// TIA Portal project "ft" (V16)

(* hardware
DEVICE "S7-1200 station_1"  S7-1200 Station
   slot 0: "Rack_0"  S7-1200 Rack  Rack  V1.0
   slot 1: "PLC_1"  CPU 1214C DC/DC/DC  6ES7 214-1AG40-0XB0  V4.2
   slot 2: "DI 16/DQ 16x24VDC_1"  6ES7 223-1BL32-0XB0  V2.0
   slot 3: "DI 16/DQ 16x24VDC_2"  6ES7 223-1BL32-0XB0  V2.0
   slot 4: "DI 16/DQ 16x24VDC_3"  6ES7 223-1BL32-0XB0  V2.0
   slot 5: "DI 16/DQ 16x24VDC_4"  6ES7 223-1BL32-0XB0  V2.0
   slot 6: "DI 16/DQ 16x24VDC_5"  6ES7 223-1BL32-0XB0  V2.0
   slot 7: "DI 16/DQ 16x24VDC_6"  6ES7 223-1BL32-0XB0  V2.0
*)

// ===== PLC "PLC_1"  CPU 1214C DC/DC/DC =====

VAR_GLOBAL   // PLC tag table "Input tags_1"
   "IN_1-0.0" AT %I0.0 : Bool;
   "IN_1-0.1" AT %I0.1 : Bool;
   "IN_1-0.2" AT %I0.2 : Bool;
   "IN_1-0.3" AT %I0.3 : Bool;
   "IN_1-0.4" AT %I0.4 : Bool;
   "IN_1-0.5" AT %I0.5 : Bool;
   "IN_1-0.6" AT %I0.6 : Bool;
   "IN_1-0.7" AT %I0.7 : Bool;
   "IN_1-1.0" AT %I1.0 : Bool;
   "IN_1-1.1" AT %I1.1 : Bool;
   "IN_1-1.2" AT %I1.5 : Bool;
   "IN_1-1.3" AT %I1.4 : Bool;
   "IN_1-1.4" AT %I1.3 : Bool;
   "IN_1-1.5" AT %I1.2 : Bool;
   "AN_1" AT %IW64 : Int;
   "AN_2" AT %IW66 : Int;
END_VAR

VAR_GLOBAL   // PLC tag table "Output tags_1"
   "OUT_1-0.0" AT %Q0.0 : Bool;
   "OUT_1-0.1" AT %Q0.1 : Bool;
   "OUT_1-0.2" AT %Q0.2 : Bool;
   "OUT_1-0.3" AT %Q0.3 : Bool;
   "OUT_1-0.4" AT %Q0.4 : Bool;
   "OUT_1-0.5" AT %Q0.5 : Bool;
   "OUT_1-0.6" AT %Q0.6 : Bool;
   "OUT_1-0.7" AT %Q0.7 : Bool;
   "OUT_1-1.0" AT %Q1.0 : Bool;
   "OUT_1-1.1" AT %Q1.1 : Bool;
END_VAR

VAR_GLOBAL   // PLC tag table "Input tags_2"
   "IN_2-0.0" AT %I8.0 : Bool;
   "IN_2-0.1" AT %I8.1 : Bool;
   "IN_2-0.2" AT %I8.2 : Bool;
   "IN_2-0.3" AT %I8.3 : Bool;
   "IN_2-0.4" AT %I8.4 : Bool;
   "IN_2-0.5" AT %I8.5 : Bool;
   "IN_2-0.6" AT %I8.6 : Bool;
   "IN_2-0.7" AT %I8.7 : Bool;
   "IN_2-1.0" AT %I9.0 : Bool;
   "IN_2-1.1" AT %I9.1 : Bool;
   "IN_2-1.2" AT %I9.2 : Bool;
   "IN_2-1.3" AT %I9.3 : Bool;
   "IN_2-1.4" AT %I9.4 : Bool;
   "IN_2-1.5" AT %I9.5 : Bool;
   "IN_2-1.6" AT %I9.6 : Bool;
   "IN_2-1.7" AT %I9.7 : Bool;
END_VAR

VAR_GLOBAL   // PLC tag table "Output tags_2"
   "OUT_2-0.0" AT %Q8.0 : Bool;
   "OUT_2-0.1" AT %Q8.1 : Bool;
   "OUT_2-0.2" AT %Q8.2 : Bool;
   "OUT_2-0.3" AT %Q8.3 : Bool;
   "OUT_2-0.4" AT %Q8.4 : Bool;
   "OUT_2-0.5" AT %Q8.5 : Bool;
   "OUT_2-0.6" AT %Q8.6 : Bool;
   "OUT_2-0.7" AT %Q8.7 : Bool;
   "OUT_2-1.0" AT %Q9.0 : Bool;
   "OUT_2-1.1" AT %Q9.1 : Bool;
   "OUT_2-1.2" AT %Q9.2 : Bool;
   "OUT_2-1.3" AT %Q9.3 : Bool;
   "OUT_2-1.4" AT %Q9.4 : Bool;
   "OUT_2-1.5" AT %Q9.5 : Bool;
   "OUT_2-1.6" AT %Q9.6 : Bool;
   "OUT_2-1.7" AT %Q9.7 : Bool;
END_VAR

VAR_GLOBAL   // PLC tag table "Input tags_3"
   "IN_3-0.0" AT %I12.0 : Bool;
   "IN_3-0.1" AT %I12.1 : Bool;
   "IN_3-0.2" AT %I12.2 : Bool;
   "IN_3-0.3" AT %I12.3 : Bool;
   "IN_3-0.4" AT %I12.4 : Bool;
   "IN_3-0.5" AT %I12.5 : Bool;
   "IN_3-0.6" AT %I12.6 : Bool;
   "IN_3-0.7" AT %I12.7 : Bool;
   "IN_3-1.0" AT %I13.0 : Bool;
   "IN_3-1.1" AT %I13.1 : Bool;
   "IN_3-1.2" AT %I13.2 : Bool;
   "IN_3-1.3" AT %I13.3 : Bool;
   "IN_3-1.4" AT %I13.4 : Bool;
   "IN_3-1.5" AT %I13.5 : Bool;
   "IN_3-1.6" AT %I13.6 : Bool;
   "IN_3-1.7" AT %I13.7 : Bool;
END_VAR

VAR_GLOBAL   // PLC tag table "Output tags_3"
   "OUT_3-0.0" AT %Q12.0 : Bool;
   "OUT_3-0.1" AT %Q12.1 : Bool;
   "OUT_3-0.2" AT %Q12.2 : Bool;
   "OUT_3-0.3" AT %Q12.3 : Bool;
   "OUT_3-0.4" AT %Q12.4 : Bool;
   "OUT_3-0.5" AT %Q12.5 : Bool;
   "OUT_3-0.6" AT %Q12.6 : Bool;
   "OUT_3-0.7" AT %Q12.7 : Bool;
   "OUT_3-1.0" AT %Q13.0 : Bool;
   "OUT_3-1.1" AT %Q13.1 : Bool;
   "OUT_3-1.2" AT %Q13.2 : Bool;
   "OUT_3-1.3" AT %Q13.3 : Bool;
   "OUT_3-1.4" AT %Q13.4 : Bool;
   "OUT_3-1.5" AT %Q13.5 : Bool;
   "OUT_3-1.6" AT %Q13.6 : Bool;
   "OUT_3-1.7" AT %Q13.7 : Bool;
END_VAR

VAR_GLOBAL   // PLC tag table "Input tags_4"
   "IN_4-0.0" AT %I16.0 : Bool;
   "IN_4-0.1" AT %I16.1 : Bool;
   "IN_4-0.2" AT %I16.2 : Bool;
   "IN_4-0.3" AT %I16.3 : Bool;
   "IN_4-0.4" AT %I16.4 : Bool;
   "IN_4-0.5" AT %I16.5 : Bool;
   "IN_4-0.6" AT %I16.6 : Bool;
   "IN_4-0.7" AT %I16.7 : Bool;
   "IN_4-1.0" AT %I17.0 : Bool;
   "IN_4-1.1" AT %I17.1 : Bool;
   "IN_4-1.2" AT %I17.2 : Bool;
   "IN_4-1.3" AT %I17.3 : Bool;
   "IN_4-1.4" AT %I17.4 : Bool;
   "IN_4-1.5" AT %I17.5 : Bool;
   "IN_4-1.6" AT %I17.6 : Bool;
   "IN_4-1.7" AT %I17.7 : Bool;
END_VAR

VAR_GLOBAL   // PLC tag table "Output tags_4"
   "OUT_4-0.0" AT %Q16.0 : Bool;
   "OUT_4-0.1" AT %Q16.1 : Bool;
   "OUT_4-0.2" AT %Q16.2 : Bool;
   "OUT_4-0.3" AT %Q16.3 : Bool;
   "OUT_4-0.4" AT %Q16.4 : Bool;
   "OUT_4-0.5" AT %Q16.5 : Bool;
   "OUT_4-0.6" AT %Q16.6 : Bool;
   "OUT_4-0.7" AT %Q16.7 : Bool;
   "OUT_4-1.0" AT %Q17.0 : Bool;
   "OUT_4-1.1" AT %Q17.1 : Bool;
   "OUT_4-1.2" AT %Q17.2 : Bool;
   "OUT_4-1.3" AT %Q17.3 : Bool;
   "OUT_4-1.4" AT %Q17.4 : Bool;
   "OUT_4-1.5" AT %Q17.5 : Bool;
   "OUT_4-1.6" AT %Q17.6 : Bool;
   "OUT_4-1.7" AT %Q17.7 : Bool;
END_VAR

VAR_GLOBAL   // PLC tag table "Input tags_5"
   "IN_5-0.0" AT %I20.0 : Bool;
   "IN_5-0.1" AT %I20.1 : Bool;
   "IN_5-0.2" AT %I20.2 : Bool;
   "IN_5-0.3" AT %I20.3 : Bool;
   "IN_5-0.4" AT %I20.4 : Bool;
   "IN_5-0.5" AT %I20.5 : Bool;
   "IN_5-0.6" AT %I20.6 : Bool;
   "IN_5-0.7" AT %I20.7 : Bool;
   "IN_5-1.0" AT %I21.0 : Bool;
   "IN_5-1.1" AT %I21.1 : Bool;
   "IN_5-1.2" AT %I21.2 : Bool;
   "IN_5-1.3" AT %I21.3 : Bool;
   "IN_5-1.4" AT %I21.4 : Bool;
   "IN_5-1.5" AT %I21.5 : Bool;
   "IN_5-1.6" AT %I21.6 : Bool;
   "IN_5-1.7" AT %I21.7 : Bool;
END_VAR

VAR_GLOBAL   // PLC tag table "Output tags_5"
   "OUT_5-0.0" AT %Q20.0 : Bool;
   "OUT_5-0.1" AT %Q20.1 : Bool;
   "OUT_5-0.2" AT %Q20.2 : Bool;
   "OUT_5-0.3" AT %Q20.3 : Bool;
   "OUT_5-0.4" AT %Q20.4 : Bool;
   "OUT_5-0.5" AT %Q20.5 : Bool;
   "OUT_5-0.6" AT %Q20.6 : Bool;
   "OUT_5-0.7" AT %Q20.7 : Bool;
   "OUT_5-1.0" AT %Q21.0 : Bool;
   "OUT_5-1.1" AT %Q21.1 : Bool;
   "OUT_5-1.2" AT %Q21.2 : Bool;
   "OUT_5-1.3" AT %Q21.3 : Bool;
   "OUT_5-1.4" AT %Q21.4 : Bool;
   "OUT_5-1.5" AT %Q21.5 : Bool;
   "OUT_5-1.6" AT %Q21.6 : Bool;
   "OUT_5-1.7" AT %Q21.7 : Bool;
END_VAR

VAR_GLOBAL   // PLC tag table "Input tags_6"
   "IN_6-0.0" AT %I24.0 : Bool;
   "IN_6-0.1" AT %I24.1 : Bool;
   "IN_6-0.2" AT %I24.2 : Bool;
   "IN_6-0.3" AT %I24.3 : Bool;
   "IN_6-0.4" AT %I24.4 : Bool;
   "IN_6-0.5" AT %I24.5 : Bool;
   "IN_6-0.6" AT %I24.6 : Bool;
   "IN_6-0.7" AT %I24.7 : Bool;
   "IN_6-1.0" AT %I25.0 : Bool;
   "IN_6-1.1" AT %I25.1 : Bool;
   "IN_6-1.2" AT %I25.2 : Bool;
   "IN_6-1.3" AT %I25.3 : Bool;
   "IN_6-1.4" AT %I25.4 : Bool;
   "IN_6-1.5" AT %I25.5 : Bool;
   "IN_6-1.6" AT %I25.6 : Bool;
   "IN_6-1.7" AT %I25.7 : Bool;
END_VAR

VAR_GLOBAL   // PLC tag table "Output tags_6"
   "OUT_6-0.0" AT %Q24.0 : Bool;
   "OUT_6-0.1" AT %Q24.1 : Bool;
   "OUT_6-0.2" AT %Q24.2 : Bool;
   "OUT_6-0.3" AT %Q24.3 : Bool;
   "OUT_6-0.4" AT %Q24.4 : Bool;
   "OUT_6-0.5" AT %Q24.5 : Bool;
   "OUT_6-0.6" AT %Q24.6 : Bool;
   "OUT_6-0.7" AT %Q24.7 : Bool;
   "OUT_6-1.0" AT %Q25.0 : Bool;
   "OUT_6-1.1" AT %Q25.1 : Bool;
   "OUT_6-1.2" AT %Q25.2 : Bool;
   "OUT_6-1.3" AT %Q25.3 : Bool;
   "OUT_6-1.4" AT %Q25.4 : Bool;
   "OUT_6-1.5" AT %Q25.5 : Bool;
   "OUT_6-1.6" AT %Q25.6 : Bool;
   "OUT_6-1.7" AT %Q25.7 : Bool;
END_VAR

VAR_GLOBAL   // PLC tag table "Input tags_7"
   "IN_7-0.0" AT %I28.0 : Bool;
   "IN_7-0.1" AT %I28.1 : Bool;
   "IN_7-0.2" AT %I28.2 : Bool;
   "IN_7-0.3" AT %I28.3 : Bool;
   "IN_7-0.4" AT %I28.4 : Bool;
   "IN_7-0.5" AT %I28.5 : Bool;
   "IN_7-0.6" AT %I28.6 : Bool;
   "IN_7-0.7" AT %I28.7 : Bool;
   "IN_7-1.0" AT %I29.0 : Bool;
   "IN_7-1.1" AT %I29.1 : Bool;
   "IN_7-1.2" AT %I29.2 : Bool;
   "IN_7-1.3" AT %I29.3 : Bool;
   "IN_7-1.4" AT %I29.4 : Bool;
   "IN_7-1.5" AT %I29.5 : Bool;
   "IN_7-1.6" AT %I29.6 : Bool;
   "IN_7-1.7" AT %I29.7 : Bool;
END_VAR

VAR_GLOBAL   // PLC tag table "Output tags_7"
   "OUT_7-0.0" AT %Q28.0 : Bool;
   "OUT_7-0.1" AT %Q28.1 : Bool;
   "OUT_7-0.2" AT %Q28.2 : Bool;
   "OUT_7-0.3" AT %Q28.3 : Bool;
   "OUT_7-0.4" AT %Q28.4 : Bool;
   "OUT_7-0.5" AT %Q28.5 : Bool;
   "OUT_7-0.6" AT %Q28.6 : Bool;
   "OUT_7-0.7" AT %Q28.7 : Bool;
   "OUT_7-1.0" AT %Q29.0 : Bool;
   "OUT_7-1.1" AT %Q29.1 : Bool;
   "OUT_7-1.2" AT %Q29.2 : Bool;
   "OUT_7-1.3" AT %Q29.3 : Bool;
   "OUT_7-1.4" AT %Q29.4 : Bool;
   "OUT_7-1.5" AT %Q29.5 : Bool;
   "OUT_7-1.6" AT %Q29.6 : Bool;
   "OUT_7-1.7" AT %Q29.7 : Bool;
END_VAR

// folder: System blocks/Program resources

DATA_BLOCK "IEC_Timer_0_DB"   // DB1
{ S7_Optimized_Access := 'TRUE' }
AUTHOR : Simatic
FAMILY : IEC
NAME : IEC_TMR
VERSION : 1.0
// stored: InstanceOfName IEC_TIMER
"IEC_TIMER"
BEGIN
END_DATA_BLOCK

DATA_BLOCK "IEC_Timer_0_DB_1"   // DB2
{ S7_Optimized_Access := 'TRUE' }
AUTHOR : Simatic
FAMILY : IEC
NAME : IEC_TMR
VERSION : 1.0
// stored: InstanceOfName IEC_TIMER
"IEC_TIMER"
BEGIN
END_DATA_BLOCK

DATA_BLOCK "IEC_Timer_0_DB_2"   // DB3
{ S7_Optimized_Access := 'TRUE' }
AUTHOR : Simatic
FAMILY : IEC
NAME : IEC_TMR
VERSION : 1.0
// stored: InstanceOfName IEC_TIMER
"IEC_TIMER"
BEGIN
END_DATA_BLOCK

DATA_BLOCK "IEC_Timer_0_DB_3"   // DB4
{ S7_Optimized_Access := 'TRUE' }
AUTHOR : Simatic
FAMILY : IEC
NAME : IEC_TMR
VERSION : 1.0
// stored: InstanceOfName IEC_TIMER
"IEC_TIMER"
BEGIN
END_DATA_BLOCK

DATA_BLOCK "IEC_Timer_0_DB_4"   // DB5
{ S7_Optimized_Access := 'TRUE' }
AUTHOR : Simatic
FAMILY : IEC
NAME : IEC_TMR
VERSION : 1.0
// stored: InstanceOfName IEC_TIMER
"IEC_TIMER"
BEGIN
END_DATA_BLOCK

DATA_BLOCK "IEC_Timer_0_DB_5"   // DB6
{ S7_Optimized_Access := 'TRUE' }
AUTHOR : Simatic
FAMILY : IEC
NAME : IEC_TMR
VERSION : 1.0
// stored: InstanceOfName IEC_TIMER
"IEC_TIMER"
BEGIN
END_DATA_BLOCK

DATA_BLOCK "IEC_Timer_0_DB_6"   // DB7
{ S7_Optimized_Access := 'TRUE' }
AUTHOR : Simatic
FAMILY : IEC
NAME : IEC_TMR
VERSION : 1.0
// stored: InstanceOfName IEC_TIMER
"IEC_TIMER"
BEGIN
END_DATA_BLOCK

DATA_BLOCK "IEC_Timer_0_DB_7"   // DB8
{ S7_Optimized_Access := 'TRUE' }
AUTHOR : Simatic
FAMILY : IEC
NAME : IEC_TMR
VERSION : 1.0
// stored: InstanceOfName IEC_TIMER
"IEC_TIMER"
BEGIN
END_DATA_BLOCK

DATA_BLOCK "IEC_Timer_0_DB_8"   // DB9
{ S7_Optimized_Access := 'TRUE' }
AUTHOR : Simatic
FAMILY : IEC
NAME : IEC_TMR
VERSION : 1.0
// stored: InstanceOfName IEC_TIMER
"IEC_TIMER"
BEGIN
END_DATA_BLOCK

DATA_BLOCK "IEC_Timer_0_DB_9"   // DB10
{ S7_Optimized_Access := 'TRUE' }
AUTHOR : Simatic
FAMILY : IEC
NAME : IEC_TMR
VERSION : 1.0
// stored: InstanceOfName IEC_TIMER
"IEC_TIMER"
BEGIN
END_DATA_BLOCK

DATA_BLOCK "IEC_Timer_0_DB_10"   // DB11
{ S7_Optimized_Access := 'TRUE' }
AUTHOR : Simatic
FAMILY : IEC
NAME : IEC_TMR
VERSION : 1.0
// stored: InstanceOfName IEC_TIMER
"IEC_TIMER"
BEGIN
END_DATA_BLOCK

DATA_BLOCK "IEC_Timer_0_DB_11"   // DB12
{ S7_Optimized_Access := 'TRUE' }
AUTHOR : Simatic
FAMILY : IEC
NAME : IEC_TMR
VERSION : 1.0
// stored: InstanceOfName IEC_TIMER
"IEC_TIMER"
BEGIN
END_DATA_BLOCK

DATA_BLOCK "IEC_Timer_0_DB_12"   // DB13
{ S7_Optimized_Access := 'TRUE' }
AUTHOR : Simatic
FAMILY : IEC
NAME : IEC_TMR
VERSION : 1.0
// stored: InstanceOfName IEC_TIMER
"IEC_TIMER"
BEGIN
END_DATA_BLOCK

DATA_BLOCK "IEC_Timer_0_DB_13"   // DB14
{ S7_Optimized_Access := 'TRUE' }
AUTHOR : Simatic
FAMILY : IEC
NAME : IEC_TMR
VERSION : 1.0
// stored: InstanceOfName IEC_TIMER
"IEC_TIMER"
BEGIN
END_DATA_BLOCK

DATA_BLOCK "IEC_Timer_0_DB_14"   // DB15
{ S7_Optimized_Access := 'TRUE' }
AUTHOR : Simatic
FAMILY : IEC
NAME : IEC_TMR
VERSION : 1.0
// stored: InstanceOfName IEC_TIMER
"IEC_TIMER"
BEGIN
END_DATA_BLOCK

DATA_BLOCK "IEC_Timer_0_DB_15"   // DB16
{ S7_Optimized_Access := 'TRUE' }
AUTHOR : Simatic
FAMILY : IEC
NAME : IEC_TMR
VERSION : 1.0
// stored: InstanceOfName IEC_TIMER
"IEC_TIMER"
BEGIN
END_DATA_BLOCK

DATA_BLOCK "IEC_Timer_0_DB_16"   // DB17
{ S7_Optimized_Access := 'TRUE' }
AUTHOR : Simatic
FAMILY : IEC
NAME : IEC_TMR
VERSION : 1.0
// stored: InstanceOfName IEC_TIMER
"IEC_TIMER"
BEGIN
END_DATA_BLOCK

DATA_BLOCK "IEC_Timer_0_DB_17"   // DB18
{ S7_Optimized_Access := 'TRUE' }
AUTHOR : Simatic
FAMILY : IEC
NAME : IEC_TMR
VERSION : 1.0
// stored: InstanceOfName IEC_TIMER
"IEC_TIMER"
BEGIN
END_DATA_BLOCK

DATA_BLOCK "IEC_Timer_0_DB_18"   // DB19
{ S7_Optimized_Access := 'TRUE' }
AUTHOR : Simatic
FAMILY : IEC
NAME : IEC_TMR
VERSION : 1.0
// stored: InstanceOfName IEC_TIMER
"IEC_TIMER"
BEGIN
END_DATA_BLOCK

DATA_BLOCK "IEC_Timer_0_DB_19"   // DB20
{ S7_Optimized_Access := 'TRUE' }
AUTHOR : Simatic
FAMILY : IEC
NAME : IEC_TMR
VERSION : 1.0
// stored: InstanceOfName IEC_TIMER
"IEC_TIMER"
BEGIN
END_DATA_BLOCK

DATA_BLOCK "IEC_Timer_0_DB_20"   // DB21
{ S7_Optimized_Access := 'TRUE' }
AUTHOR : Simatic
FAMILY : IEC
NAME : IEC_TMR
VERSION : 1.0
// stored: InstanceOfName IEC_TIMER
"IEC_TIMER"
BEGIN
END_DATA_BLOCK

DATA_BLOCK "IEC_Timer_0_DB_21"   // DB22
{ S7_Optimized_Access := 'TRUE' }
AUTHOR : Simatic
FAMILY : IEC
NAME : IEC_TMR
VERSION : 1.0
// stored: InstanceOfName IEC_TIMER
"IEC_TIMER"
BEGIN
END_DATA_BLOCK

DATA_BLOCK "IEC_Timer_0_DB_22"   // DB23
{ S7_Optimized_Access := 'TRUE' }
AUTHOR : Simatic
FAMILY : IEC
NAME : IEC_TMR
VERSION : 1.0
// stored: InstanceOfName IEC_TIMER
"IEC_TIMER"
BEGIN
END_DATA_BLOCK

DATA_BLOCK "IEC_Timer_0_DB_23"   // DB24
{ S7_Optimized_Access := 'TRUE' }
AUTHOR : Simatic
FAMILY : IEC
NAME : IEC_TMR
VERSION : 1.0
// stored: InstanceOfName IEC_TIMER
"IEC_TIMER"
BEGIN
END_DATA_BLOCK

DATA_BLOCK "IEC_Timer_0_DB_24"   // DB25
{ S7_Optimized_Access := 'TRUE' }
AUTHOR : Simatic
FAMILY : IEC
NAME : IEC_TMR
VERSION : 1.0
// stored: InstanceOfName IEC_TIMER
"IEC_TIMER"
BEGIN
END_DATA_BLOCK

DATA_BLOCK "IEC_Timer_0_DB_25"   // DB26
{ S7_Optimized_Access := 'TRUE' }
AUTHOR : Simatic
FAMILY : IEC
NAME : IEC_TMR
VERSION : 1.0
// stored: InstanceOfName IEC_TIMER
"IEC_TIMER"
BEGIN
END_DATA_BLOCK

DATA_BLOCK "IEC_Timer_0_DB_26"   // DB27
{ S7_Optimized_Access := 'TRUE' }
AUTHOR : Simatic
FAMILY : IEC
NAME : IEC_TMR
VERSION : 1.0
// stored: InstanceOfName IEC_TIMER
"IEC_TIMER"
BEGIN
END_DATA_BLOCK

DATA_BLOCK "IEC_Timer_0_DB_27"   // DB28
{ S7_Optimized_Access := 'TRUE' }
AUTHOR : Simatic
FAMILY : IEC
NAME : IEC_TMR
VERSION : 1.0
// stored: InstanceOfName IEC_TIMER
"IEC_TIMER"
BEGIN
END_DATA_BLOCK

DATA_BLOCK "IEC_Timer_0_DB_28"   // DB29
{ S7_Optimized_Access := 'TRUE' }
AUTHOR : Simatic
FAMILY : IEC
NAME : IEC_TMR
VERSION : 1.0
// stored: InstanceOfName IEC_TIMER
"IEC_TIMER"
BEGIN
END_DATA_BLOCK

DATA_BLOCK "IEC_Timer_0_DB_29"   // DB30
{ S7_Optimized_Access := 'TRUE' }
AUTHOR : Simatic
FAMILY : IEC
NAME : IEC_TMR
VERSION : 1.0
// stored: InstanceOfName IEC_TIMER
"IEC_TIMER"
BEGIN
END_DATA_BLOCK

DATA_BLOCK "IEC_Timer_0_DB_30"   // DB31
{ S7_Optimized_Access := 'TRUE' }
AUTHOR : Simatic
FAMILY : IEC
NAME : IEC_TMR
VERSION : 1.0
// stored: InstanceOfName IEC_TIMER
"IEC_TIMER"
BEGIN
END_DATA_BLOCK

DATA_BLOCK "IEC_Timer_0_DB_31"   // DB32
{ S7_Optimized_Access := 'TRUE' }
AUTHOR : Simatic
FAMILY : IEC
NAME : IEC_TMR
VERSION : 1.0
// stored: InstanceOfName IEC_TIMER
"IEC_TIMER"
BEGIN
END_DATA_BLOCK

DATA_BLOCK "IEC_Timer_0_DB_32"   // DB33
{ S7_Optimized_Access := 'TRUE' }
AUTHOR : Simatic
FAMILY : IEC
NAME : IEC_TMR
VERSION : 1.0
// stored: InstanceOfName IEC_TIMER
"IEC_TIMER"
BEGIN
END_DATA_BLOCK

DATA_BLOCK "IEC_Timer_0_DB_33"   // DB34
{ S7_Optimized_Access := 'TRUE' }
AUTHOR : Simatic
FAMILY : IEC
NAME : IEC_TMR
VERSION : 1.0
// stored: InstanceOfName IEC_TIMER
"IEC_TIMER"
BEGIN
END_DATA_BLOCK

DATA_BLOCK "IEC_Timer_0_DB_34"   // DB35
{ S7_Optimized_Access := 'TRUE' }
AUTHOR : Simatic
FAMILY : IEC
NAME : IEC_TMR
VERSION : 1.0
// stored: InstanceOfName IEC_TIMER
"IEC_TIMER"
BEGIN
END_DATA_BLOCK

DATA_BLOCK "IEC_Timer_0_DB_35"   // DB36
{ S7_Optimized_Access := 'TRUE' }
AUTHOR : Simatic
FAMILY : IEC
NAME : IEC_TMR
VERSION : 1.0
// stored: InstanceOfName IEC_TIMER
"IEC_TIMER"
BEGIN
END_DATA_BLOCK

DATA_BLOCK "IEC_Timer_0_DB_36"   // DB37
{ S7_Optimized_Access := 'TRUE' }
AUTHOR : Simatic
FAMILY : IEC
NAME : IEC_TMR
VERSION : 1.0
// stored: InstanceOfName IEC_TIMER
"IEC_TIMER"
BEGIN
END_DATA_BLOCK

DATA_BLOCK "IEC_Timer_0_DB_37"   // DB38
{ S7_Optimized_Access := 'TRUE' }
AUTHOR : Simatic
FAMILY : IEC
NAME : IEC_TMR
VERSION : 1.0
// stored: InstanceOfName IEC_TIMER
"IEC_TIMER"
BEGIN
END_DATA_BLOCK

// folder: (top level)

ORGANIZATION_BLOCK "Main"   // OB1, LAD, ProgramCycle
TITLE = "Main Program Sweep (Cycle)"
{ S7_Optimized_Access := 'TRUE' }
VERSION : 0.1
   VAR_INPUT
      Initial_Call : Bool;   // Initial call of this OB
      Remanence : Bool;   // =True, if remanent data are available
   END_VAR
   VAR CONSTANT
      T1 : Time := T#2500ms;
      T2 : Time := T#1200ms;
      T3 : Time := T#2275ms;
      T4 : Time := T#100ms;
      T5 : Time := T#3000ms;
      T6 : Time := T#1500ms;
      T7 : Time := T#2000ms;
      T8 : Time := T#800ms;
      T9 : Time := T#3500ms;
      T10 : Time := T#1390ms;
      T11 : Time := T#25000ms;
      T12 : Time := T#500ms;
   END_VAR
BEGIN

REGION Network 1
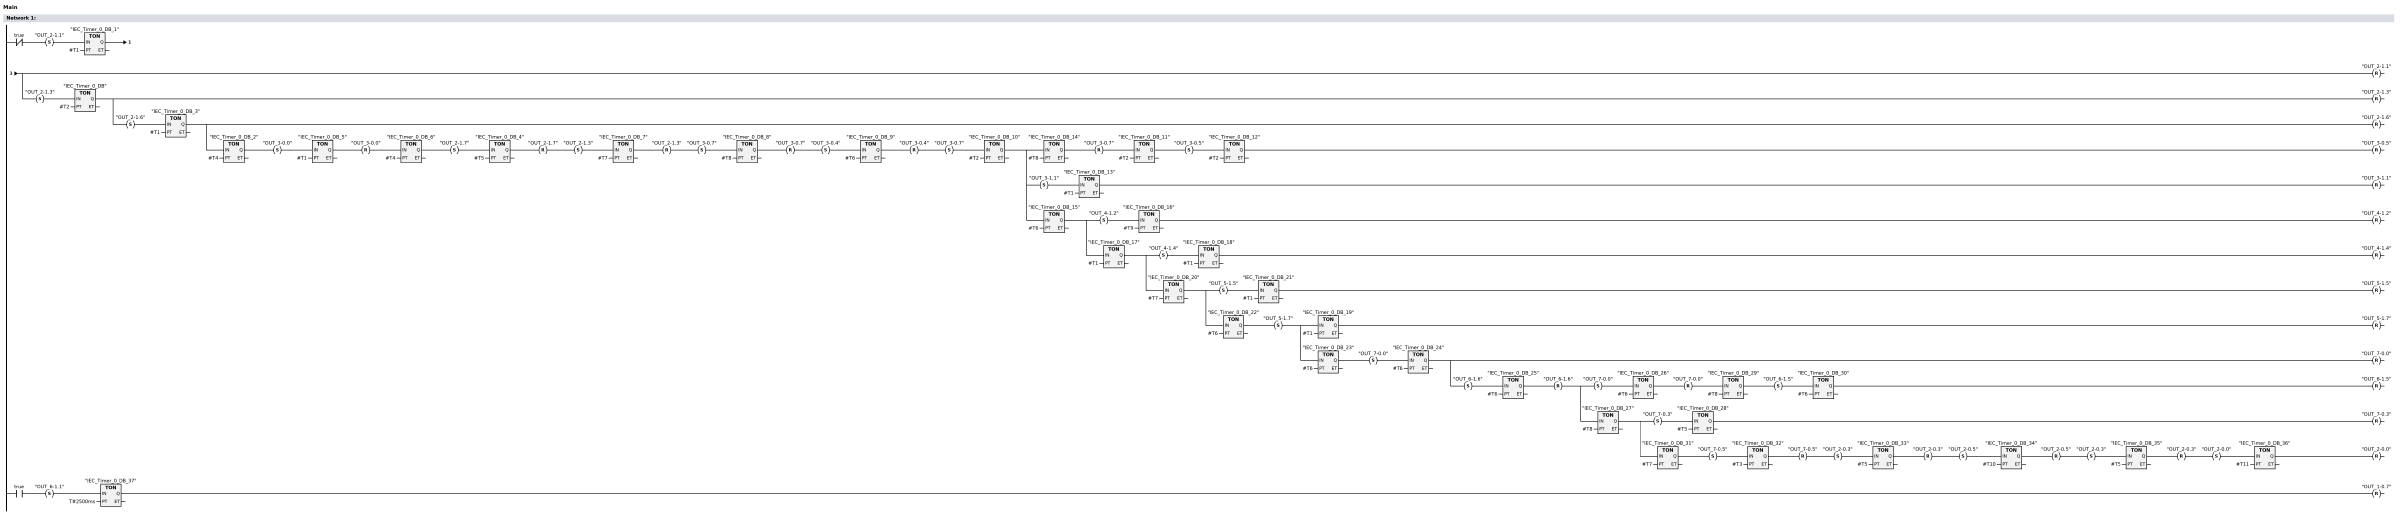
   IF NOT true THEN "OUT_2-1.1" := TRUE; END_IF;
   "IEC_Timer_0_DB_1".TON(IN := NOT true, PT := #T1);
   IF "IEC_Timer_0_DB_1".Q THEN
       "OUT_2-1.1" := FALSE;
       "OUT_2-1.3" := TRUE;
   END_IF;
   "IEC_Timer_0_DB".TON(IN := "IEC_Timer_0_DB_1".Q, PT := #T2);
   IF "IEC_Timer_0_DB".Q THEN
       "OUT_2-1.3" := FALSE;
       "OUT_2-1.6" := TRUE;
   END_IF;
   "IEC_Timer_0_DB_3".TON(IN := "IEC_Timer_0_DB".Q, PT := #T1);
   IF "IEC_Timer_0_DB_3".Q THEN "OUT_2-1.6" := FALSE; END_IF;
   "IEC_Timer_0_DB_2".TON(IN := "IEC_Timer_0_DB_3".Q, PT := #T4);
   IF "IEC_Timer_0_DB_2".Q THEN "OUT_3-0.0" := TRUE; END_IF;
   "IEC_Timer_0_DB_5".TON(IN := "IEC_Timer_0_DB_2".Q, PT := #T1);
   IF "IEC_Timer_0_DB_5".Q THEN "OUT_3-0.0" := FALSE; END_IF;
   "IEC_Timer_0_DB_6".TON(IN := "IEC_Timer_0_DB_5".Q, PT := #T4);
   IF "IEC_Timer_0_DB_6".Q THEN "OUT_2-1.7" := TRUE; END_IF;
   "IEC_Timer_0_DB_4".TON(IN := "IEC_Timer_0_DB_6".Q, PT := #T5);
   IF "IEC_Timer_0_DB_4".Q THEN
       "OUT_2-1.7" := FALSE;
       "OUT_2-1.3" := TRUE;
   END_IF;
   "IEC_Timer_0_DB_7".TON(IN := "IEC_Timer_0_DB_4".Q, PT := #T7);
   IF "IEC_Timer_0_DB_7".Q THEN
       "OUT_2-1.3" := FALSE;
       "OUT_3-0.7" := TRUE;
   END_IF;
   "IEC_Timer_0_DB_8".TON(IN := "IEC_Timer_0_DB_7".Q, PT := #T8);
   IF "IEC_Timer_0_DB_8".Q THEN
       "OUT_3-0.7" := FALSE;
       "OUT_3-0.4" := TRUE;
   END_IF;
   "IEC_Timer_0_DB_9".TON(IN := "IEC_Timer_0_DB_8".Q, PT := #T6);
   IF "IEC_Timer_0_DB_9".Q THEN
       "OUT_3-0.4" := FALSE;
       "OUT_3-0.7" := TRUE;
   END_IF;
   "IEC_Timer_0_DB_10".TON(IN := "IEC_Timer_0_DB_9".Q, PT := #T2);
   "IEC_Timer_0_DB_14".TON(IN := "IEC_Timer_0_DB_10".Q, PT := #T8);
   IF "IEC_Timer_0_DB_14".Q THEN "OUT_3-0.7" := FALSE; END_IF;
   "IEC_Timer_0_DB_11".TON(IN := "IEC_Timer_0_DB_14".Q, PT := #T2);
   IF "IEC_Timer_0_DB_11".Q THEN "OUT_3-0.5" := TRUE; END_IF;
   "IEC_Timer_0_DB_12".TON(IN := "IEC_Timer_0_DB_11".Q, PT := #T2);
   IF "IEC_Timer_0_DB_12".Q THEN "OUT_3-0.5" := FALSE; END_IF;
   IF "IEC_Timer_0_DB_10".Q THEN "OUT_3-1.1" := TRUE; END_IF;
   "IEC_Timer_0_DB_13".TON(IN := "IEC_Timer_0_DB_10".Q, PT := #T1);
   IF "IEC_Timer_0_DB_13".Q THEN "OUT_3-1.1" := FALSE; END_IF;
   "IEC_Timer_0_DB_15".TON(IN := "IEC_Timer_0_DB_10".Q, PT := #T6);
   IF "IEC_Timer_0_DB_15".Q THEN "OUT_4-1.2" := TRUE; END_IF;
   "IEC_Timer_0_DB_16".TON(IN := "IEC_Timer_0_DB_15".Q, PT := #T9);
   IF "IEC_Timer_0_DB_16".Q THEN "OUT_4-1.2" := FALSE; END_IF;
   "IEC_Timer_0_DB_17".TON(IN := "IEC_Timer_0_DB_15".Q, PT := #T1);
   IF "IEC_Timer_0_DB_17".Q THEN "OUT_4-1.4" := TRUE; END_IF;
   "IEC_Timer_0_DB_18".TON(IN := "IEC_Timer_0_DB_17".Q, PT := #T1);
   IF "IEC_Timer_0_DB_18".Q THEN "OUT_4-1.4" := FALSE; END_IF;
   "IEC_Timer_0_DB_20".TON(IN := "IEC_Timer_0_DB_17".Q, PT := #T7);
   IF "IEC_Timer_0_DB_20".Q THEN "OUT_5-1.5" := TRUE; END_IF;
   "IEC_Timer_0_DB_21".TON(IN := "IEC_Timer_0_DB_20".Q, PT := #T1);
   IF "IEC_Timer_0_DB_21".Q THEN "OUT_5-1.5" := FALSE; END_IF;
   "IEC_Timer_0_DB_22".TON(IN := "IEC_Timer_0_DB_20".Q, PT := #T6);
   IF "IEC_Timer_0_DB_22".Q THEN "OUT_5-1.7" := TRUE; END_IF;
   "IEC_Timer_0_DB_19".TON(IN := "IEC_Timer_0_DB_22".Q, PT := #T1);
   IF "IEC_Timer_0_DB_19".Q THEN "OUT_5-1.7" := FALSE; END_IF;
   "IEC_Timer_0_DB_23".TON(IN := "IEC_Timer_0_DB_22".Q, PT := #T6);
   IF "IEC_Timer_0_DB_23".Q THEN "OUT_7-0.0" := TRUE; END_IF;
   "IEC_Timer_0_DB_24".TON(IN := "IEC_Timer_0_DB_23".Q, PT := #T6);
   IF "IEC_Timer_0_DB_24".Q THEN
       "OUT_7-0.0" := FALSE;
       "OUT_6-1.6" := TRUE;
   END_IF;
   "IEC_Timer_0_DB_25".TON(IN := "IEC_Timer_0_DB_24".Q, PT := #T6);
   IF "IEC_Timer_0_DB_25".Q THEN
       "OUT_6-1.6" := FALSE;
       "OUT_7-0.0" := TRUE;
   END_IF;
   "IEC_Timer_0_DB_26".TON(IN := "IEC_Timer_0_DB_25".Q, PT := #T6);
   IF "IEC_Timer_0_DB_26".Q THEN "OUT_7-0.0" := FALSE; END_IF;
   "IEC_Timer_0_DB_29".TON(IN := "IEC_Timer_0_DB_26".Q, PT := #T8);
   IF "IEC_Timer_0_DB_29".Q THEN "OUT_6-1.5" := TRUE; END_IF;
   "IEC_Timer_0_DB_30".TON(IN := "IEC_Timer_0_DB_29".Q, PT := #T6);
   IF "IEC_Timer_0_DB_30".Q THEN "OUT_6-1.5" := FALSE; END_IF;
   "IEC_Timer_0_DB_27".TON(IN := "IEC_Timer_0_DB_25".Q, PT := #T8);
   IF "IEC_Timer_0_DB_27".Q THEN "OUT_7-0.3" := TRUE; END_IF;
   "IEC_Timer_0_DB_28".TON(IN := "IEC_Timer_0_DB_27".Q, PT := #T5);
   IF "IEC_Timer_0_DB_28".Q THEN "OUT_7-0.3" := FALSE; END_IF;
   "IEC_Timer_0_DB_31".TON(IN := "IEC_Timer_0_DB_27".Q, PT := #T7);
   IF "IEC_Timer_0_DB_31".Q THEN "OUT_7-0.5" := TRUE; END_IF;
   "IEC_Timer_0_DB_32".TON(IN := "IEC_Timer_0_DB_31".Q, PT := #T3);
   IF "IEC_Timer_0_DB_32".Q THEN
       "OUT_7-0.5" := FALSE;
       "OUT_2-0.3" := TRUE;
   END_IF;
   "IEC_Timer_0_DB_33".TON(IN := "IEC_Timer_0_DB_32".Q, PT := #T5);
   IF "IEC_Timer_0_DB_33".Q THEN
       "OUT_2-0.3" := FALSE;
       "OUT_2-0.5" := TRUE;
   END_IF;
   "IEC_Timer_0_DB_34".TON(IN := "IEC_Timer_0_DB_33".Q, PT := #T10);
   IF "IEC_Timer_0_DB_34".Q THEN
       "OUT_2-0.5" := FALSE;
       "OUT_2-0.3" := TRUE;
   END_IF;
   "IEC_Timer_0_DB_35".TON(IN := "IEC_Timer_0_DB_34".Q, PT := #T5);
   IF "IEC_Timer_0_DB_35".Q THEN
       "OUT_2-0.3" := FALSE;
       "OUT_2-0.0" := TRUE;
   END_IF;
   "IEC_Timer_0_DB_36".TON(IN := "IEC_Timer_0_DB_35".Q, PT := #T11);
   IF "IEC_Timer_0_DB_36".Q THEN "OUT_2-0.0" := FALSE; END_IF;
   IF true THEN "OUT_6-1.1" := TRUE; END_IF;
   "IEC_Timer_0_DB_37".TON(IN := true, PT := T#2500ms);
   IF "IEC_Timer_0_DB_37".Q THEN "OUT_1-0.7" := FALSE; END_IF;
END_REGION
END_ORGANIZATION_BLOCK